(********************* G.D S.p.A. - Technical Department ***********************************
This program has been generated automatically from Application Designer DE&F
********************************************************************************************)
PROGRAM dbg_csp_case_transport_ls_trailing
VAR
  axis_shd : axis_shadow;
END_VAR

_objects_manager();

IF	g_application_status <> APPLICATION_STATUS_RUNNING
THEN
	RETURN;
END_IF

CASE process_get_mode(CONVERSION_this := dbg_root.prc) OF
	MODE_ABSENT,
	MODE_INACTIVE:
		RETURN;
	MODE_TEST:
		RETURN;
END_CASE

ACTION _objects_manager:
IF	objects_initialization()
THEN
	axis_shadow_init(
		sim_mode:= SHADOW_SIMULATION_MODE_AUTOMATIC, 
		father:= csp_case_transport_ls_trailing.axis, 
		process:= dbg_root.prc, 
		CONVERSION_this:= axis_shd);

	RETURN;
END_IF

IF	objects_running()
THEN
	axis_shadow_cycle(axis_shd);
END_IF
END_ACTION

END_PROGRAM

(* stored: Version 1.1.0.1, ProductVersion 3.1.4022.12
   POU dbg_csp_case_transport_ls_trailing: Id {078c5314-bff8-4b70-a819-3b9c103794f7}, SpecialFunc None
   Action _objects_manager: Id {f853b26c-92a5-412f-897b-a4209ca889e0} *)
